FUNCTION_BLOCK PML_Method_Base
VAR_INPUT
END_VAR
VAR_OUTPUT
END_VAR
VAR
	ipackml : IPmlStateMachine;
END_VAR

CASE ipackml.GetCurrentState() OF
	E_PMLState.ePMLState_Clearing:
		Clearing();
	E_PMLState.ePMLState_Aborted:
		Aborted();
	E_PMLState.ePMLState_Aborting:
		Aborting();
	E_PMLState.ePMLState_Complete:
		Completed();
	E_PMLState.ePMLState_Completing:
		Completing();
	E_PMLState.ePMLState_Execute:
		Execute();
	E_PMLState.ePMLState_Held:
		Held();
	E_PMLState.ePMLState_Holding:
		Holding();
	E_PMLState.ePMLState_Idle:
		Idle();
	E_PMLState.ePMLState_Resetting:
		Resetting();
	E_PMLState.ePMLState_Starting:
		Starting();
	E_PMLState.ePMLState_Stopped:
		Stopped();
	E_PMLState.ePMLState_Stopping:
		Stopping();
	E_PMLState.ePMLState_Suspended:
		Suspended();
	E_PMLState.ePMLState_Suspending:
		Suspending();
	E_PMLState.ePMLState_Undefined:
		Undefined();
	E_PMLState.ePMLState_Unholding:
		Unholding();
	E_PMLState.ePMLState_Unsuspending:
		Unsuspending();
END_CASE

METHOD PRIVATE Aborted : BOOL
VAR_INPUT
END_VAR
END_METHOD

METHOD PRIVATE Aborting : BOOL
VAR_INPUT
END_VAR
ipackml.SetStateComplete();
END_METHOD

METHOD PRIVATE Clearing : BOOL
VAR_INPUT
END_VAR
ipackml.SetStateComplete();
END_METHOD

METHOD PRIVATE Completed : BOOL
VAR_INPUT
END_VAR
END_METHOD

METHOD PRIVATE Completing : BOOL
VAR_INPUT
END_VAR
ipackml.SetStateComplete();
END_METHOD

METHOD PRIVATE Execute : BOOL
VAR_INPUT
END_VAR
END_METHOD

METHOD PRIVATE Held : BOOL
VAR_INPUT
END_VAR
END_METHOD

METHOD PRIVATE Holding : BOOL
VAR_INPUT
END_VAR
ipackml.SetStateComplete();
END_METHOD

METHOD PRIVATE Idle : BOOL
VAR_INPUT
END_VAR
END_METHOD

PROPERTY PUBLIC PackMLStateMachine : IPmlStateMachine
GET
PackMLStateMachine := ipackml;
END_GET
SET
ipackml := PackMLStateMachine;
END_SET
END_PROPERTY

METHOD PRIVATE Resetting : BOOL
VAR_INPUT
END_VAR
ipackml.SetStateComplete();
END_METHOD

METHOD PRIVATE Starting : BOOL
VAR_INPUT
END_VAR
ipackml.SetStateComplete();
END_METHOD

METHOD PRIVATE Stopped : BOOL
VAR_INPUT
END_VAR
END_METHOD

METHOD PRIVATE Stopping : BOOL
VAR_INPUT
END_VAR
ipackml.SetStateComplete();
END_METHOD

METHOD PRIVATE Suspended : BOOL
VAR_INPUT
END_VAR
END_METHOD

METHOD PRIVATE Suspending : BOOL
VAR_INPUT
END_VAR
ipackml.SetStateComplete();
END_METHOD

METHOD PRIVATE Undefined : BOOL
VAR_INPUT
END_VAR
END_METHOD

METHOD PRIVATE Unholding : BOOL
VAR_INPUT
END_VAR
ipackml.SetStateComplete();
END_METHOD

METHOD PRIVATE Unsuspending : BOOL
VAR_INPUT
END_VAR
ipackml.SetStateComplete();
END_METHOD

END_FUNCTION_BLOCK

(* stored: Version 1.1.0.1, ProductVersion 3.1.4024.11
   POU PML_Method_Base: Id {e9cf9054-9269-474f-9eb2-f1589d2b309b}, SpecialFunc None
   Folder Action_States: Id {b5e75466-7e20-4308-9a0c-d79f927f78b2}
   Folder Wait_States: Id {4ea05185-b1a4-4062-8470-b5d9cd15033c}
   Method Aborted: Id {0b53e203-5e54-4083-a358-85f9fcb0b82d}
   Method Aborting: Id {a238d54d-264d-44d5-8ffa-3c1950f83c82}
   Method Clearing: Id {bc0d4280-1f13-44f7-9829-54e43797220d}
   Method Completed: Id {a2cdb556-85a9-4482-9c68-efa360a9f3a8}
   Method Completing: Id {d000f392-3ce7-4095-9ef8-8fd0d9356f52}
   Method Execute: Id {c7bd509a-3b83-4cba-a198-2c15be7394c6}
   Method Held: Id {43527c9b-adbe-4a8d-bea9-48bd143c16e1}
   Method Holding: Id {51b21d7c-d045-491a-9230-89c46c7877ba}
   Method Idle: Id {72ae97ce-bb49-416c-a0c3-2a5d5a89b363}
   Property PackMLStateMachine: Id {cf5e7a1b-4ee5-46c8-9a79-b6965176ee5b}
   Get Get: Id {dec79564-8f21-411e-afc4-a59804408c09}
   Set Set: Id {22e113bd-b318-41f5-8eea-5dd3d4547564}
   Method Resetting: Id {a2baa753-5fca-484b-ac9d-210e1d858721}
   Method Starting: Id {7130edc4-9bcd-4f22-a7e3-a08ef79934ac}
   Method Stopped: Id {9216c521-0aa8-4d36-b21b-e92e18d080de}
   Method Stopping: Id {d1deb6dc-cf14-43e2-9c49-5843d0609c07}
   Method Suspended: Id {3a3bac37-3c3e-4d16-8e35-91a2f397e3f4}
   Method Suspending: Id {2c5d472d-4db0-4bfa-8212-c6994a3a3a1e}
   Method Undefined: Id {c2968a58-cc56-487d-837d-e21cd9003270}
   Method Unholding: Id {c38e73f1-8378-4b42-b35b-fb73989464ff}
   Method Unsuspending: Id {d39bdcd4-1b3a-4864-8589-79f8ff046f53} *)
